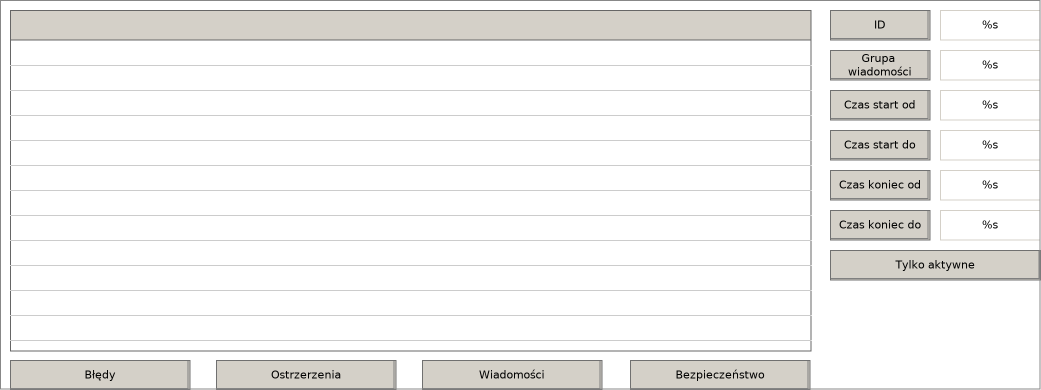
VISUALIZATION Visu_LogowanieBledow_Tabela  // 1041x390
VAR_IN_OUT
	stParametry								: DUT_LogowanieBledow_WyswietlanieParametry;
END_VAR
    Table (10,10 801x341), data array: GVL_LogowanieBledow.fbLoger.arrTablicaWyswietlana
        p3854506369: GVL_LogowanieBledow.fbLoger.arrTablicaWyswietlana[INDEX].sNrKomponentu
        p1892666644: GVL_LogowanieBledow.fbLoger.arrTablicaWyswietlana[INDEX].sKodBledu
        p338671338: GVL_LogowanieBledow.fbLoger.arrTablicaWyswietlana[INDEX].byRodzajZdarzenia
        p2170511999: GVL_LogowanieBledow.fbLoger.arrTablicaWyswietlana[INDEX].sOpis
        p3723444502: GVL_LogowanieBledow.fbLoger.arrTablicaWyswietlana[INDEX].dtDataStart
        p1218418051: GVL_LogowanieBledow.fbLoger.arrTablicaWyswietlana[INDEX].dtDataKoniec
        p746581629: GVL_LogowanieBledow.fbLoger.arrTablicaWyswietlana[INDEX].dwKolor
        p2232123230: Nr Elem.
        p2237128397: Data start
        p505689113: Data koniec
    Button (830,10 100x30), "ID", colour toggle: stParametry.bFiltrID
        toggle stParametry.bFiltrID
    Button (830,50 100x30), "Grupa wiadomości", colour toggle: stParametry.bFiltrRodzaj
        toggle stParametry.bFiltrRodzaj
    Button (830,90 100x30), "Czas start od", colour toggle: stParametry.bFiltrStartOD
        toggle stParametry.bFiltrStartOD
    Button (830,130 100x30), "Czas start do", colour toggle: stParametry.bFiltrStartDO
        toggle stParametry.bFiltrStartDO
    Button (830,170 100x30), "Czas koniec od", colour toggle: stParametry.bFiltrKoniecOD
        toggle stParametry.bFiltrKoniecOD
    Button (830,210 100x30), "Czas koniec do", colour toggle: stParametry.bFiltrKoniecDO
        toggle stParametry.bFiltrKoniecDO
    Button (830,250 211x30), "Tylko aktywne", colour toggle: stParametry.bFiltrAktywne
        toggle stParametry.bFiltrAktywne
    Textfield (940,10 100x30), "%s", text variable: stParametry.iFiltrID
        OnMouseDown: write the text variable via VisuDialogs.Numpad
    Textfield (940,50 100x30), "%s", text variable: stParametry.byFiltrRodzaj
        OnMouseDown: write the text variable via VisuDialogs.Numpad
    Textfield (940,90 100x30), "%s", text variable: stParametry.dtFiltrStartOD
        OnMouseDown: write the text variable via Edit
    Textfield (940,130 100x30), "%s", text variable: stParametry.dtFiltrStartDO
        OnMouseDown: write the text variable via Edit
    Textfield (940,170 100x30), "%s", text variable: stParametry.dtFiltrKoniecOD
        OnMouseDown: write the text variable via Edit
    Textfield (940,210 100x30), "%s", text variable: stParametry.dtFiltrKoniecDO
        OnMouseDown: write the text variable via Edit
    Button (10,360 180x30), "Błędy", colour toggle: stParametry.bFiltrRodzaj and stParametry.byFiltrRodzaj = 1
        OnMouseDown: execute {
            IF (NOT stParametry.bFiltrRodzaj) THEN
            	stParametry.bFiltrRodzaj := TRUE;
            	stParametry.byFiltrRodzaj := 1;
            ELSE
            	stParametry.bFiltrRodzaj := FALSE;
            END_IF
        }
    Button (216,360 180x30), "Ostrzerzenia", colour toggle: stParametry.bFiltrRodzaj and stParametry.byFiltrRodzaj = 2
        OnMouseDown: execute {
            IF (NOT stParametry.bFiltrRodzaj) THEN
            	stParametry.bFiltrRodzaj := TRUE;
            	stParametry.byFiltrRodzaj := 2;
            ELSE
            	stParametry.bFiltrRodzaj := FALSE;
            END_IF
        }
    Button (422,360 180x30), "Wiadomości", colour toggle: stParametry.bFiltrRodzaj and stParametry.byFiltrRodzaj = 3
        OnMouseDown: execute {
            IF (NOT stParametry.bFiltrRodzaj) THEN
            	stParametry.bFiltrRodzaj := TRUE;
            	stParametry.byFiltrRodzaj := 3;
            ELSE
            	stParametry.bFiltrRodzaj := FALSE;
            END_IF
        }
    Button (630,360 180x30), "Bezpieczeństwo", colour toggle: stParametry.bFiltrRodzaj and stParametry.byFiltrRodzaj = 4
        OnMouseDown: execute {
            IF (NOT stParametry.bFiltrRodzaj) THEN
            	stParametry.bFiltrRodzaj := TRUE;
            	stParametry.byFiltrRodzaj := 4;
            ELSE
            	stParametry.bFiltrRodzaj := FALSE;
            END_IF
        }
END_VISUALIZATION

(* stored: Version 1.1.0.1, ProductVersion 3.1.4024.11
   Visu Visu_LogowanieBledow_Tabela: Id {3dc9ce44-38c3-4cfe-98bb-3fc546ae08da} *)
